{attribute 'qualified_only'}
{attribute 'strict'}
TYPE E_AREA :
(
	NotDef := 0,
	OpenArea := 1,
	ConstrainedArea := 2,
	PrakingArea := 3,
	LoadArea := 4
);
END_TYPE

(* stored: Version 1.1.0.1, ProductVersion 3.1.4024.11
   DUT E_AREA: Id {387797d1-7c26-4554-8660-3baa32342ed8} *)
